INTERFACE I_NciCommand EXTENDS I_Command

END_INTERFACE

(* stored: Version 1.1.0.1, ProductVersion 3.1.4024.12
   Itf I_NciCommand: Id {7003bd1e-bc6c-48f8-b72b-0c829271f0bf} *)
